PROGRAM MAIN
VAR
	FB_SyncrhonousTest : FB_SyncrhonousTest;
END_VAR

FB_SyncrhonousTest();

END_PROGRAM

(* stored: Version 1.1.0.1
   POU MAIN: Id {7534196b-5208-4624-b3e1-4d0093be325e}, SpecialFunc None *)
